{attribute addProperty BoxType "EL5152-0000-0016"}
{attribute addProperty Id "Period_valueAT %I*UDINT324"}
{attribute addProperty CRC "2891036832"}
{attribute addProperty SizeInBites "32"}
{attribute addProperty SizeInBytes "4"}
TYPE ENC_Period_Channel_AC51B8A0 :
STRUCT
	{attribute addProperty Name "Period_value"}
	Period_value AT %I* : UDINT;
END_STRUCT
END_TYPE

(* stored: Version 1.2.0.0, ProductVersion 3.1.4024.9
   DUT ENC_Period_Channel_AC51B8A0: Id {e8cfc3e7-30c4-4e0c-933d-168cf5c8b6fa} *)
